PROGRAM TEST_PRG
VAR
END_VAR

TcUnit.RUN();

END_PROGRAM

(* stored: Version 1.1.0.1, ProductVersion 3.1.4024.12
   POU TEST_PRG: Id {f82fcdb8-2c22-4362-bb6e-b02954d36a8d}, SpecialFunc None *)
